// TIA Portal V17 export
// export: Created 2022-03-12T16:05:31.4284412Z, ExportSetting WithDefaults, DisplayName Totally Integrated Automation Portal, DisplayVersion V17, DisplayName TIA Portal Openness, DisplayVersion V17, DisplayName TIA Portal Version Control Interface, DisplayVersion V17, DisplayName STEP 7 Professional, DisplayVersion V17, DisplayName STEP 7 Safety, DisplayVersion V17, DisplayName WinCC Advanced / Unified PC, DisplayVersion V17
DATA_BLOCK "HMI_Data_Custom"   // DB31616
TITLE = CPG_HMI_Data_Custom
{ S7_Optimized_Access := 'TRUE' }
AUTHOR : tech.team.motioncontrol@siemens.com
FAMILY : CPG
VERSION : 1.0
// Support: tech.team.motioncontrol@siemens.com
// Fax: +49 (0) 9131/98-1297
// stored: AutoNumber true, DBAccessibleFromOPCUA true, DBAccessibleFromWebserver true, IsOnlyStoredInLoadMemory false, IsRetainMemResEnabled false, IsWriteProtectedInAS false, MemoryReserve 0
   VAR
      machineSpeedSP : Real := 20.0;   // Machine Speed Setpoint (product per min)
      machineSpeedPV { ExternalWritable := 'False'} : Real;   // Machine Speed Actual (product per min)
   END_VAR
BEGIN
END_DATA_BLOCK
